// TIA Portal project "双数码管显示学号_蔡文嘉_V14" (V14)

(* hardware
DEVICE "S7-1200 station_1"  S7-1200 Station
   slot 0: "Rack_0"  Rack  V1.0
DEVICE "S7-1200 station_2"  S7-1200 Station
   slot 0: "Rack_0"  Rack  V1.0
   slot 1: "PLC_1"  CPU 1214C DC/DC/DC  6ES7 214-1AG40-0XB0  V4.1
DEVICE "HMI_1"  KTP700 Basic PN
   slot 0: "HMI"  HMI  6AV2 123-2GB03-0AX0  13.0.1.0
   slot 1: "HMI_RT_1"  KTP700 Basic PN  6AV2 123-2GB03-0AX0  13.0.1.0
   slot 5: "HMI_1.IE_CP_1"  PROFINET 接口
      slot 1: "PROFINET Interface_1"  PROFINET 接口
         slot 1: "Port_1"  端口
*)

// ===== PLC "PLC_1"  CPU 1214C DC/DC/DC =====

VAR_GLOBAL   // PLC tag table "默认变量表"
   "启动" AT %M0.0 : Bool;
   "停止" AT %M0.1 : Bool;
   "自动计数开始" AT %M0.2 : Bool;
   "A" AT %Q0.0 : Bool;
   "B" AT %Q0.1 : Bool;
   "C" AT %Q0.2 : Bool;
   "D" AT %Q0.3 : Bool;
   "E" AT %Q0.4 : Bool;
   "F" AT %Q0.5 : Bool;
   "G" AT %Q0.6 : Bool;
   "LED显示数字" AT %MW10 : Word;
   "LED数码管16进制段位" AT %QB0 : Byte;
   "A1" AT %Q1.0 : Bool;
   "B1" AT %Q1.1 : Bool;
   "C1" AT %Q1.2 : Bool;
   "D1" AT %Q1.3 : Bool;
   "E1" AT %Q1.4 : Bool;
   "F1" AT %Q1.5 : Bool;
   "G1" AT %Q1.6 : Bool;
   "LED显示数字1" AT %MW20 : Word;
   "LED数码管16进制段位1" AT %QB1 : Byte;
END_VAR

// folder: System blocks/Program resources

DATA_BLOCK "Timer_10"   // DB1
{ S7_Optimized_Access := 'TRUE' }
AUTHOR : Simatic
FAMILY : IEC
NAME : IEC_TMR
VERSION : 1.0
// stored: InstanceOfName IEC_TIMER
"IEC_TIMER"
BEGIN
END_DATA_BLOCK

DATA_BLOCK "Timer_2"   // DB3
{ S7_Optimized_Access := 'TRUE' }
AUTHOR : Simatic
FAMILY : IEC
NAME : IEC_TMR
VERSION : 1.0
// stored: InstanceOfName IEC_TIMER
"IEC_TIMER"
BEGIN
END_DATA_BLOCK

DATA_BLOCK "Timer_3"   // DB4
{ S7_Optimized_Access := 'TRUE' }
AUTHOR : Simatic
FAMILY : IEC
NAME : IEC_TMR
VERSION : 1.0
// stored: InstanceOfName IEC_TIMER
"IEC_TIMER"
BEGIN
END_DATA_BLOCK

DATA_BLOCK "Timer_4"   // DB5
{ S7_Optimized_Access := 'TRUE' }
AUTHOR : Simatic
FAMILY : IEC
NAME : IEC_TMR
VERSION : 1.0
// stored: InstanceOfName IEC_TIMER
"IEC_TIMER"
BEGIN
END_DATA_BLOCK

DATA_BLOCK "Timer_5"   // DB6
{ S7_Optimized_Access := 'TRUE' }
AUTHOR : Simatic
FAMILY : IEC
NAME : IEC_TMR
VERSION : 1.0
// stored: InstanceOfName IEC_TIMER
"IEC_TIMER"
BEGIN
END_DATA_BLOCK

DATA_BLOCK "Timer_6"   // DB7
{ S7_Optimized_Access := 'TRUE' }
AUTHOR : Simatic
FAMILY : IEC
NAME : IEC_TMR
VERSION : 1.0
// stored: InstanceOfName IEC_TIMER
"IEC_TIMER"
BEGIN
END_DATA_BLOCK

DATA_BLOCK "Timer_7"   // DB8
{ S7_Optimized_Access := 'TRUE' }
AUTHOR : Simatic
FAMILY : IEC
NAME : IEC_TMR
VERSION : 1.0
// stored: InstanceOfName IEC_TIMER
"IEC_TIMER"
BEGIN
END_DATA_BLOCK

DATA_BLOCK "Timer_8"   // DB9
{ S7_Optimized_Access := 'TRUE' }
AUTHOR : Simatic
FAMILY : IEC
NAME : IEC_TMR
VERSION : 1.0
// stored: InstanceOfName IEC_TIMER
"IEC_TIMER"
BEGIN
END_DATA_BLOCK

DATA_BLOCK "Timer_9"   // DB10
{ S7_Optimized_Access := 'TRUE' }
AUTHOR : Simatic
FAMILY : IEC
NAME : IEC_TMR
VERSION : 1.0
// stored: InstanceOfName IEC_TIMER
"IEC_TIMER"
BEGIN
END_DATA_BLOCK

DATA_BLOCK "Timer_11"   // DB11
{ S7_Optimized_Access := 'TRUE' }
AUTHOR : Simatic
FAMILY : IEC
NAME : IEC_TMR
VERSION : 1.0
// stored: InstanceOfName IEC_TIMER
"IEC_TIMER"
BEGIN
END_DATA_BLOCK

// folder: (top level)

ORGANIZATION_BLOCK "Main"   // OB1, LAD, ProgramCycle
TITLE = "Main Program Sweep (Cycle)"
{ S7_Optimized_Access := 'TRUE' }
VERSION : 0.1
   VAR_INPUT
      Initial_Call : Bool;   // Initial call of this OB
      Remanence : Bool;   // =True, if remanent data are available
   END_VAR
BEGIN

REGION Network 1
   // 启动、停止操作
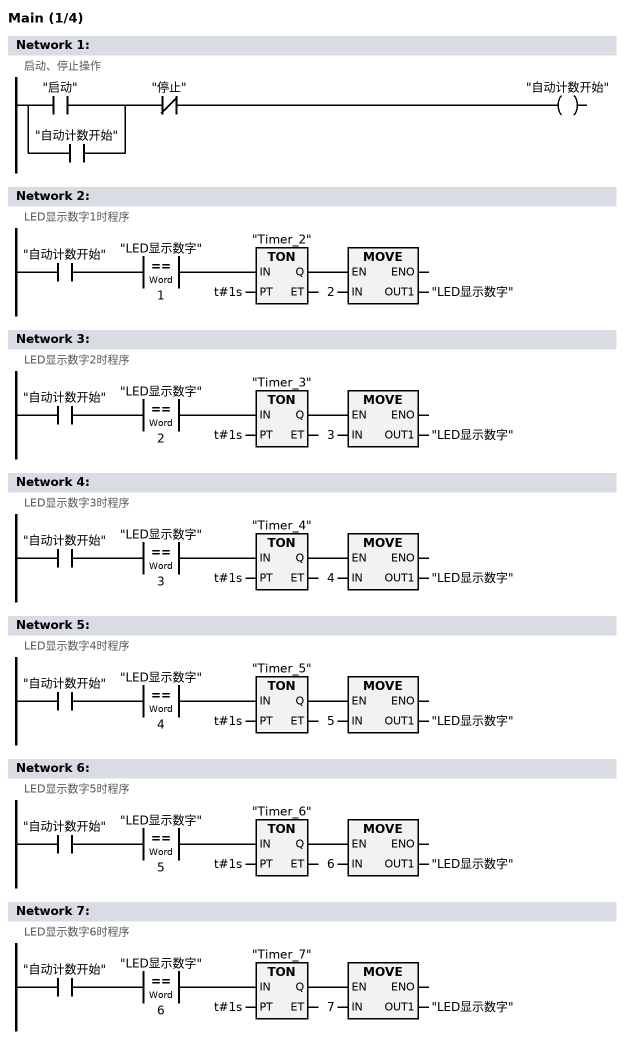
   RUNG wire#powerrail
      Contact( "启动" )
      wire#w1
      I_Contact( "停止" )
      Coil( "自动计数开始" )
   END_RUNG
   RUNG wire#powerrail
      Contact( "自动计数开始" )
   END_RUNG wire#w1
   // the same network as SCL:
   "自动计数开始" := ("启动" OR "自动计数开始") AND NOT "停止";
END_REGION

REGION Network 2
   // LED显示数字1时程序
   "Timer_2".TON(IN := "自动计数开始" AND ("LED显示数字" = 1), PT := t#1s);
   IF "Timer_2".Q THEN "LED显示数字" := 2; END_IF;
END_REGION

REGION Network 3
   // LED显示数字2时程序
   "Timer_3".TON(IN := "自动计数开始" AND ("LED显示数字" = 2), PT := t#1s);
   IF "Timer_3".Q THEN "LED显示数字" := 3; END_IF;
END_REGION

REGION Network 4
   // LED显示数字3时程序
   "Timer_4".TON(IN := "自动计数开始" AND ("LED显示数字" = 3), PT := t#1s);
   IF "Timer_4".Q THEN "LED显示数字" := 4; END_IF;
END_REGION

REGION Network 5
   // LED显示数字4时程序
   "Timer_5".TON(IN := "自动计数开始" AND ("LED显示数字" = 4), PT := t#1s);
   IF "Timer_5".Q THEN "LED显示数字" := 5; END_IF;
END_REGION

REGION Network 6
   // LED显示数字5时程序
   "Timer_6".TON(IN := "自动计数开始" AND ("LED显示数字" = 5), PT := t#1s);
   IF "Timer_6".Q THEN "LED显示数字" := 6; END_IF;
END_REGION

REGION Network 7
   // LED显示数字6时程序
   "Timer_7".TON(IN := "自动计数开始" AND ("LED显示数字" = 6), PT := t#1s);
   IF "Timer_7".Q THEN "LED显示数字" := 7; END_IF;
END_REGION

REGION Network 8
   // LED显示数字7时程序
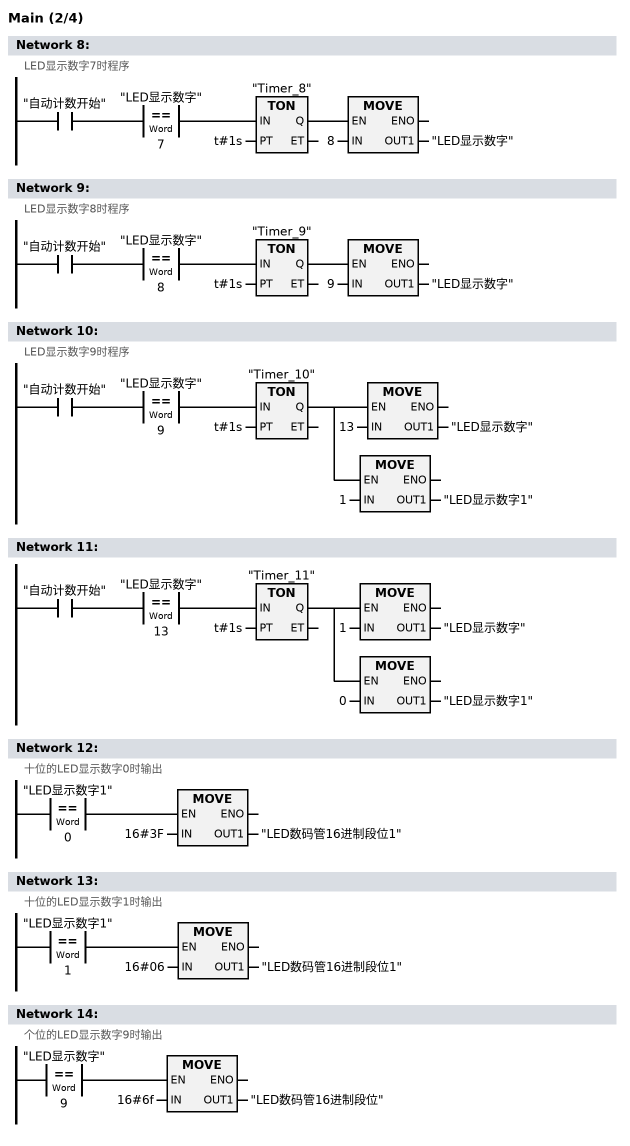
   "Timer_8".TON(IN := "自动计数开始" AND ("LED显示数字" = 7), PT := t#1s);
   IF "Timer_8".Q THEN "LED显示数字" := 8; END_IF;
END_REGION

REGION Network 9
   // LED显示数字8时程序
   "Timer_9".TON(IN := "自动计数开始" AND ("LED显示数字" = 8), PT := t#1s);
   IF "Timer_9".Q THEN "LED显示数字" := 9; END_IF;
END_REGION

REGION Network 10
   // LED显示数字9时程序
   "Timer_10".TON(IN := "自动计数开始" AND ("LED显示数字" = 9), PT := t#1s);
   IF "Timer_10".Q THEN
       "LED显示数字" := 13;
       "LED显示数字1" := 1;
   END_IF;
END_REGION

REGION Network 11
   "Timer_11".TON(IN := "自动计数开始" AND ("LED显示数字" = 13), PT := t#1s);
   IF "Timer_11".Q THEN
       "LED显示数字" := 1;
       "LED显示数字1" := 0;
   END_IF;
END_REGION

REGION Network 12
   // 十位的LED显示数字0时输出
   RUNG wire#powerrail
      { S7_Templates := "SrcType := Word" } EQ_Contact(in1 := "LED显示数字1", in2 := 0)
      Move(in := 16#3F, out1 => "LED数码管16进制段位1")
   END_RUNG
   // the same network as SCL:
   IF "LED显示数字1" = 0 THEN "LED数码管16进制段位1" := 16#3F; END_IF;
END_REGION

REGION Network 13
   // 十位的LED显示数字1时输出
   RUNG wire#powerrail
      { S7_Templates := "SrcType := Word" } EQ_Contact(in1 := "LED显示数字1", in2 := 1)
      Move(in := 16#06, out1 => "LED数码管16进制段位1")
   END_RUNG
   // the same network as SCL:
   IF "LED显示数字1" = 1 THEN "LED数码管16进制段位1" := 16#06; END_IF;
END_REGION

REGION Network 14
   // 个位的LED显示数字9时输出
   RUNG wire#powerrail
      { S7_Templates := "SrcType := Word" } EQ_Contact(in1 := "LED显示数字", in2 := 9)
      Move(in := 16#6f, out1 => "LED数码管16进制段位")
   END_RUNG
   // the same network as SCL:
   IF "LED显示数字" = 9 THEN "LED数码管16进制段位" := 16#6f; END_IF;
END_REGION

REGION Network 15
   // 个位的LED显示数字1时输出
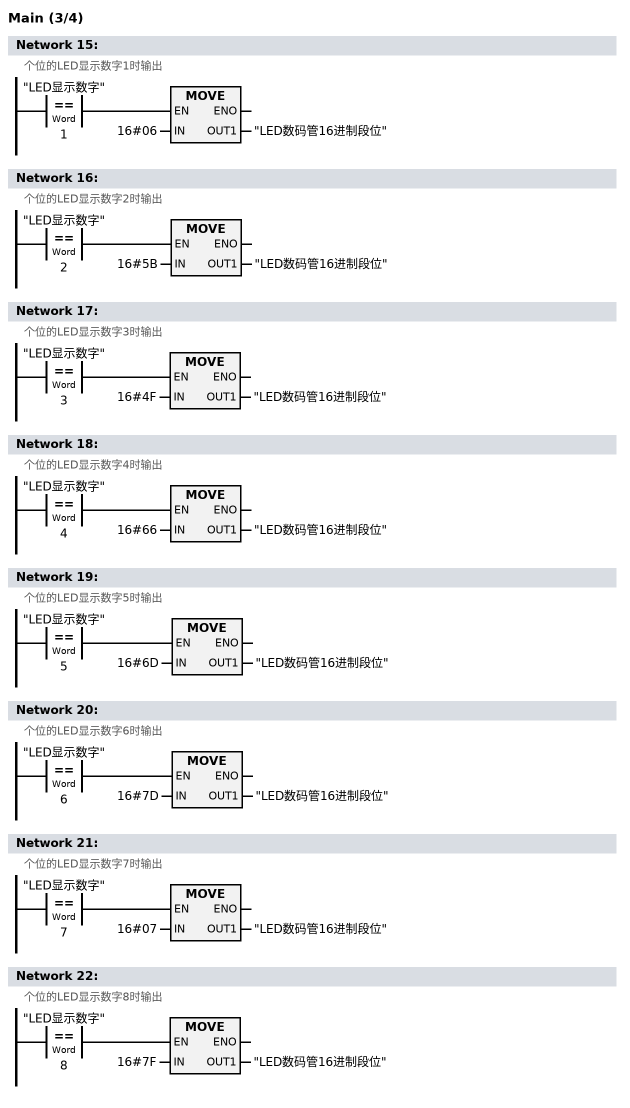
   RUNG wire#powerrail
      { S7_Templates := "SrcType := Word" } EQ_Contact(in1 := "LED显示数字", in2 := 1)
      Move(in := 16#06, out1 => "LED数码管16进制段位")
   END_RUNG
   // the same network as SCL:
   IF "LED显示数字" = 1 THEN "LED数码管16进制段位" := 16#06; END_IF;
END_REGION

REGION Network 16
   // 个位的LED显示数字2时输出
   RUNG wire#powerrail
      { S7_Templates := "SrcType := Word" } EQ_Contact(in1 := "LED显示数字", in2 := 2)
      Move(in := 16#5B, out1 => "LED数码管16进制段位")
   END_RUNG
   // the same network as SCL:
   IF "LED显示数字" = 2 THEN "LED数码管16进制段位" := 16#5B; END_IF;
END_REGION

REGION Network 17
   // 个位的LED显示数字3时输出
   RUNG wire#powerrail
      { S7_Templates := "SrcType := Word" } EQ_Contact(in1 := "LED显示数字", in2 := 3)
      Move(in := 16#4F, out1 => "LED数码管16进制段位")
   END_RUNG
   // the same network as SCL:
   IF "LED显示数字" = 3 THEN "LED数码管16进制段位" := 16#4F; END_IF;
END_REGION

REGION Network 18
   // 个位的LED显示数字4时输出
   RUNG wire#powerrail
      { S7_Templates := "SrcType := Word" } EQ_Contact(in1 := "LED显示数字", in2 := 4)
      Move(in := 16#66, out1 => "LED数码管16进制段位")
   END_RUNG
   // the same network as SCL:
   IF "LED显示数字" = 4 THEN "LED数码管16进制段位" := 16#66; END_IF;
END_REGION

REGION Network 19
   // 个位的LED显示数字5时输出
   RUNG wire#powerrail
      { S7_Templates := "SrcType := Word" } EQ_Contact(in1 := "LED显示数字", in2 := 5)
      Move(in := 16#6D, out1 => "LED数码管16进制段位")
   END_RUNG
   // the same network as SCL:
   IF "LED显示数字" = 5 THEN "LED数码管16进制段位" := 16#6D; END_IF;
END_REGION

REGION Network 20
   // 个位的LED显示数字6时输出
   RUNG wire#powerrail
      { S7_Templates := "SrcType := Word" } EQ_Contact(in1 := "LED显示数字", in2 := 6)
      Move(in := 16#7D, out1 => "LED数码管16进制段位")
   END_RUNG
   // the same network as SCL:
   IF "LED显示数字" = 6 THEN "LED数码管16进制段位" := 16#7D; END_IF;
END_REGION

REGION Network 21
   // 个位的LED显示数字7时输出
   RUNG wire#powerrail
      { S7_Templates := "SrcType := Word" } EQ_Contact(in1 := "LED显示数字", in2 := 7)
      Move(in := 16#07, out1 => "LED数码管16进制段位")
   END_RUNG
   // the same network as SCL:
   IF "LED显示数字" = 7 THEN "LED数码管16进制段位" := 16#07; END_IF;
END_REGION

REGION Network 22
   // 个位的LED显示数字8时输出
   RUNG wire#powerrail
      { S7_Templates := "SrcType := Word" } EQ_Contact(in1 := "LED显示数字", in2 := 8)
      Move(in := 16#7F, out1 => "LED数码管16进制段位")
   END_RUNG
   // the same network as SCL:
   IF "LED显示数字" = 8 THEN "LED数码管16进制段位" := 16#7F; END_IF;
END_REGION

REGION Network 23
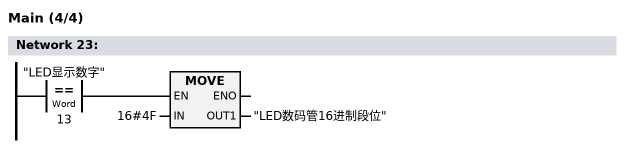
   RUNG wire#powerrail
      { S7_Templates := "SrcType := Word" } EQ_Contact(in1 := "LED显示数字", in2 := 13)
      Move(in := 16#4F, out1 => "LED数码管16进制段位")
   END_RUNG
   // the same network as SCL:
   IF "LED显示数字" = 13 THEN "LED数码管16进制段位" := 16#4F; END_IF;
END_REGION
END_ORGANIZATION_BLOCK

(* ===== HMI "HMI_RT_1" =====
system functions are stored by id; their names below are inferred from use
connection "HMI_连接_1": ETHERNET, SMART_S7_1200_OMS

HMI tags "默认变量表"
   "Tag_ScreenNumber" : UInt, internal
   "A" : Bool = PLC A AT %Q0.0, 1 s
   "B" : Bool = PLC B AT %Q0.1, 1 s
   "C" : Bool = PLC C AT %Q0.2, 1 s
   "D" : Bool = PLC D AT %Q0.3, 1 s
   "E" : Bool = PLC E AT %Q0.4, 1 s
   "F" : Bool = PLC F AT %Q0.5, 1 s
   "G" : Bool = PLC G AT %Q0.6, 1 s
   "启动" : Bool = PLC 启动 AT %M0.0, 1 s
   "停止" : Bool = PLC 停止 AT %M0.1, 1 s
   "LED显示数字" : Word = PLC LED显示数字 AT %MW10, 1 s
   "A1" : Bool = PLC A1 AT %Q1.0, 1 s
   "B1" : Bool = PLC B1 AT %Q1.1, 1 s
   "C1" : Bool = PLC C1 AT %Q1.2, 1 s
   "D1" : Bool = PLC D1 AT %Q1.3, 1 s
   "E1" : Bool = PLC E1 AT %Q1.4, 1 s
   "F1" : Bool = PLC F1 AT %Q1.5, 1 s
   "G1" : Bool = PLC G1 AT %Q1.6, 1 s

Template "Template_1" 800x480
   Button "Template_Button" at 714,429 size 71x50; TextOff 'ExitRuntime'; PictureOff "ExitRuntime_KTP700_Basic_PN_TR"; PictureOn "ExitRuntime_KTP700_Basic_PN_TR"
      on Release: StopRuntime(0)
   Button "Template_Button_1" at 614,429 size 71x50; TextOff 'Text'
   Button "Template_Button_2" at 514,429 size 71x50; TextOff 'Text'
   Button "Template_Button_3" at 414,429 size 71x50; TextOff 'Text'
   Button "Template_Button_4" at 314,429 size 71x50; TextOff 'Text'
   Button "Template_Button_5" at 214,429 size 71x50; TextOff 'Text'
   Button "Template_Button_6" at 114,429 size 71x50; TextOff 'AlarmDisplay'; PictureOff "AlarmDisplay_KTP700_Basic_PN_TR"; PictureOn "AlarmDisplay_KTP700_Basic_PN_TR"
      on Release: function_ef3f5d25("报警窗口_Unacknowledged", -1)
   Button "Template_Button_7" at 14,429 size 71x50; TextOff 'NavigateHome'; PictureOff "NavigateHome_KTP700_Basic_PN_TR"; PictureOn "NavigateHome_KTP700_Basic_PN_TR"
      on Release: ActivateScreen("根画面", 0)
   SymbolicIOField "Symbolic_IO_Field_Screen" at 93,9 size 600x33; TextOff '0'; TextOn '1'; TextList "TextList_ScreenNames"
      ProcessValue <- "Tag_ScreenNumber"
      on Change: ActivateScreenByNumber("Tag_ScreenNumber", 0)
   DateTimeField "HmiScreenItemData" at 695,25 size 105x25
   DateTimeField "HmiScreenItemData_1" at 695,0 size 105x25
   GraphicView "Logo" at 0,0 size 91x51; Picture "HMI_1 的 Logo"

screen "根画面" 800x480, template "Template_1"
   on GenerateScreen: SetTag("Tag_ScreenNumber", 1)
   TextField "HmiScreenItemData" at 80,228 size 640x25; Text '欢迎进入 HMI_1 (KTP700 Basic+ PN)！'

screen "自动计数" 800x480
   Rectangle "矩形_1" at 346,91 size 96x17
      Appearance <- "A"
   Rectangle "矩形_2" at 442,216 size 17x96
      Appearance <- "C"
   Rectangle "矩形_3" at 330,107 size 17x96
      Appearance <- "F"
   Rectangle "矩形_4" at 346,199 size 96x17
      Appearance <- "G"
   Rectangle "矩形_5" at 330,216 size 17x96
      Appearance <- "E"
   Rectangle "矩形_6" at 442,107 size 17x96
      Appearance <- "B"
   Rectangle "矩形_7" at 347,312 size 96x17
      Appearance <- "D"
   TextField "文本域_1" at 381,58 size 14x20; Text 'a'
   TextField "文本域_2" at 464,130 size 14x20; Text 'b'
   TextField "文本域_3" at 464,259 size 14x20; Text 'c'
   TextField "文本域_4" at 381,288 size 14x20; Text 'd'
   TextField "文本域_5" at 304,130 size 14x20; Text 'f'
   TextField "文本域_6" at 304,268 size 14x20; Text 'e'
   TextField "文本域_8" at 381,173 size 14x20; Text 'g'
   Button "按钮_1" at 613,58 size 96x32; TextOff '启动'
      on Press: SetBit("启动")
      on Release: ResetBit("启动")
   Button "按钮_2" at 612,104 size 96x32; TextOff '停止'
      on Release: ResetBit("停止")
      on Press: SetBit("停止")
   IOField "I/O 域_1" at 656,203 size 94x48; FormatPattern 99
      ProcessValue <- "LED显示数字"
   TextField "文本域_7" at 555,216 size 90x20; Text '手动输入：'
   Rectangle "矩形_8" at 164,92 size 96x17
      Appearance <- "A1"
   Rectangle "矩形_9" at 260,217 size 17x96
      Appearance <- "C1"
   Rectangle "矩形_10" at 148,108 size 17x96
      Appearance <- "F1"
   Rectangle "矩形_11" at 164,200 size 96x17
      Appearance <- "G1"
   Rectangle "矩形_12" at 148,217 size 17x96
      Appearance <- "E1"
   Rectangle "矩形_13" at 260,108 size 17x96
      Appearance <- "B1"
   Rectangle "矩形_14" at 165,313 size 96x17
      Appearance <- "D1"
   TextField "文本域_9" at 199,59 size 23x20; Text 'a1'
   TextField "文本域_10" at 277,153 size 23x20; Text 'b1'
   TextField "文本域_11" at 277,251 size 23x20; Text 'c1'
   TextField "文本域_12" at 199,289 size 23x20; Text 'd1'
   TextField "文本域_13" at 122,131 size 23x20; Text 'f1'
   TextField "文本域_14" at 122,260 size 23x20; Text 'e1'
   TextField "文本域_15" at 199,174 size 23x20; Text 'g1'
*)